FUNCTION LIMIT : DINT
	VAR_INPUT
		MN : DINT;
		IN : DINT;
		MX : DINT;
	END_VAR
BEGIN
	IF IN < MN THEN
		LIMIT := MN;
	ELSIF IN > MX THEN
		LIMIT := MX;
	ELSE
		LIMIT := MN;
	END_IF;
END_FUNCTION

FUNCTION_BLOCK STACK_DINT
	VAR_INPUT
		PUSH : BOOL;
		POP  : BOOL;
		R1   : BOOL;
		IN   : DINT;
		N    : DINT;
	END_VAR
	VAR_OUTPUT
		EMPTY : BOOL := TRUE;
		OFLO  : BOOL := FALSE;
		OUT   : DINT := 0;
		SIZE  : DINT;
	END_VAR
	VAR
		STK : ARRAY [0 .. 9] OF DINT;
		NI  : DINT := 10;
		PTR : DINT := -1;
	END_VAR
BEGIN
	IF R1 THEN
		OFLO := 0;
		EMPTY := 1;
		PTR := -1;
		NI := LIMIT(
			MN := 1,
			IN := N,
			MX := 128
		);
		OUT := 0;
	ELSIF POP & NOT EMPTY THEN
		OFLO := 0;
		PTR := PTR - 1;
		EMPTY := PTR < 0;

		IF EMPTY THEN
			OUT := 0;
		ELSE
			CASE PTR OF
				0:
					OUT := STK[0];
				1:
					OUT := STK[1];
				2:
					OUT := STK[2];
				3:
					OUT := STK[3];
				4:
					OUT := STK[4];
				5:
					OUT := STK[5];
				6:
					OUT := STK[6];
				7:
					OUT := STK[7];
				8:
					OUT := STK[8];
				9:
					OUT := STK[9];
			END_CASE;
		END_IF;
	ELSIF PUSH & NOT OFLO THEN
		EMPTY := 0;
		PTR := PTR + 1;
		OFLO := (PTR = NI);

		IF NOT OFLO THEN
			OUT := IN;
			CASE PTR OF
				0:
					STK[0] := IN;
				1:
					STK[1] := IN;
				2:
					STK[2] := IN;
				3:
					STK[3] := IN;
				4:
					STK[4] := IN;
				5:
					STK[5] := IN;
				6:
					STK[6] := IN;
				7:
					STK[7] := IN;
				8:
					STK[8] := IN;
				9:
					STK[9] := IN;
			END_CASE;
		ELSE
			OUT := 0;
		END_IF;
	END_IF;

END_FUNCTION_BLOCK

PROGRAM Main
	VAR
		I1           : DINT;
		I2           : DINT;
		I3           : DINT;
		I4           : DINT;
		B1           : BOOL;
		B2           : BOOL;
		B3           : BOOL;
		STACK_INT_FB : STACK_DINT;
		STACKOUT     : DINT;
		STACKEMPTY   : BOOL;
		STACKFULL    : BOOL;
		STACKSIZE    : DINT;
		CYCLE        : DINT := 0;
	END_VAR
BEGIN
	CYCLE := CYCLE + 1;
	STACK_INT_FB(
		PUSH := B1,
		POP := B2,
		R1 := B3,
		IN := I1,
		N := I2
	);
	STACKOUT := STACK_INT_FB.OUT;
	STACKEMPTY := STACK_INT_FB.EMPTY;
	STACKFULL := STACK_INT_FB.OFLO;
	STACKSIZE := STACK_INT_FB.SIZE;
END_PROGRAM

